{attribute 'Tc2GvlVarNames'}
{attribute 'strict'}
TYPE e_ProgrammiMovimentoY :
(
	
	Y_PosDiRiposo						:= 0,
	Y_PosFuoriIngombroRiposo 			:= 6,

	Y_PosPrelievoFalda					:= 51,
	Y_PosDepositoSuCatastaFalda			:= 52,
	Y_PosDepositoFalda					:= 53,
	//Y_PosDepositoInLentaFalda			:= 55,
	Y_PosFuoriIngombroVuotoFalda 		:= 56,
	Y_PosFuoriIngombroCaricoFalda		:= 66,

	Y_PosStartLentaPrelievoLastra 		:= 101,
	Y_PosPrelievoInLentaLastra 			:= 102,
	Y_PosDistaccoLastraInLentaLastra	:= 103,
	Y_PosStartLentaDepositoLastra 		:= 104,
	Y_PosDepositoInLentaLastra			:= 105,
	Y_PosFuoriIngombroVuotoLastra		:= 106,
	Y_PosFuoriIngombroCaricoLastra		:= 126,
	Y_PosgiroPieza						:= 127,
	Y_PosPasillo0grados					:= 128,
	Y_PosPasillo180grados				:= 129
);
END_TYPE

(* stored: Version 1.1.0.1, ProductVersion 3.1.4024.11
   EnumerationTextList e_ProgrammiMovimentoY: Id {2d232fc5-20a9-4367-96d1-d7afb4802316} *)
